{attribute addProperty BoxType "EL6224-0000-0016"}
{attribute addProperty Id "DeviceState_InputsAT %I*DeviceState_Inputs_BDC6BEC33240IO_Inputs_ChannelARRAY[0..3] OF EMPTY_STRUCTURE000IO_Outputs_ChannelARRAY[0..3] OF EMPTY_STRUCTURE000WcStateAT %I*WcState_F855686C1620InfoDataAT %I*InfoData_275E3363128160"}
{attribute addProperty CRC "2985772541"}
{attribute addProperty SizeInBites "176"}
{attribute addProperty SizeInBytes "22"}
TYPE EL6224_CC9621B7 :
STRUCT
	{attribute addProperty Name "DeviceState_Inputs"}
	DeviceState_Inputs : DeviceState_Inputs_BDC6BEC3;
	{attribute addProperty Name "IO_Inputs_Channel"}
	IO_Inputs_Channel : ARRAY[0..3] OF EMPTY_STRUCTURE;
	{attribute addProperty Name "IO_Outputs_Channel"}
	IO_Outputs_Channel : ARRAY[0..3] OF EMPTY_STRUCTURE;
	{attribute addProperty Name "WcState"}
	WcState : WcState_F855686C;
	{attribute addProperty Name "InfoData"}
	InfoData : InfoData_275E3363;
END_STRUCT
END_TYPE

(* stored: Version 1.2.0.0, ProductVersion 3.1.4024.9
   DUT EL6224_CC9621B7: Id {4f14dc8c-6b81-4576-b693-62e744b4cb24} *)
